(* CoDeSys 2.3 export: MID3.EXP *)

(* POU Mathematical/MID3, ST *)
FUNCTION MID3 : REAL
VAR_INPUT
	IN1 : REAL;
	IN2 : REAL;
	IN3 : REAL;
END_VAR


(*
version 1.2	18. mar. 2011
programmer 	hugo
tested by		tobias

returns the mid value of 3 real inputs.

*)
IF IN1 > IN2 THEN MID3 := IN1; IN1 := IN2; IN2 := MID3; END_IF;
IF IN2 > IN3 THEN IN2 := IN3; END_IF;
MID3 := SEL(IN1 > IN2, IN2, IN1);


(*
hm	1.1.2007	rev 1.1
	rewrote the function for better performance

hm	18. mar. 2011	rev 1.2
	improve performance
*)
END_FUNCTION
